GLOBALCONSTANTS DefaultPool_PI_Bargraph (* Bargraph geometry and scale constants (Length, ScalePx, Min, Max, Type) *)
  PACKAGE Uebungen::const::UT::PI;
  VAR_GLOBAL CONSTANT
    Bargraph_PI_I01_ScalePx : REAL := 4.68;
    Bargraph_PI_I01_LengthPx : REAL := 468.0;
    Bargraph_PI_I01_Min : REAL := 0.0;
    Bargraph_PI_I01_Max : REAL := 100.0;
    Bargraph_PI_I01_Type : USINT := 3;
    Bargraph_PI_I02_ScalePx : REAL := 4.68;
    Bargraph_PI_I02_LengthPx : REAL := 468.0;
    Bargraph_PI_I02_Min : REAL := 0.0;
    Bargraph_PI_I02_Max : REAL := 100.0;
    Bargraph_PI_I02_Type : USINT := 3;
    Bargraph_PI_I03_ScalePx : REAL := 4.68;
    Bargraph_PI_I03_LengthPx : REAL := 468.0;
    Bargraph_PI_I03_Min : REAL := 0.0;
    Bargraph_PI_I03_Max : REAL := 100.0;
    Bargraph_PI_I03_Type : USINT := 3;
    Bargraph_PI_I04_ScalePx : REAL := 4.68;
    Bargraph_PI_I04_LengthPx : REAL := 468.0;
    Bargraph_PI_I04_Min : REAL := 0.0;
    Bargraph_PI_I04_Max : REAL := 100.0;
    Bargraph_PI_I04_Type : USINT := 3;
    Bargraph_PI_I05_ScalePx : REAL := 4.68;
    Bargraph_PI_I05_LengthPx : REAL := 468.0;
    Bargraph_PI_I05_Min : REAL := 0.0;
    Bargraph_PI_I05_Max : REAL := 100.0;
    Bargraph_PI_I05_Type : USINT := 3;
    Bargraph_PI_I06_ScalePx : REAL := 4.68;
    Bargraph_PI_I06_LengthPx : REAL := 468.0;
    Bargraph_PI_I06_Min : REAL := 0.0;
    Bargraph_PI_I06_Max : REAL := 100.0;
    Bargraph_PI_I06_Type : USINT := 3;
    Bargraph_PI_I07_ScalePx : REAL := 4.68;
    Bargraph_PI_I07_LengthPx : REAL := 468.0;
    Bargraph_PI_I07_Min : REAL := 0.0;
    Bargraph_PI_I07_Max : REAL := 100.0;
    Bargraph_PI_I07_Type : USINT := 3;
    Bargraph_PI_I08_ScalePx : REAL := 4.68;
    Bargraph_PI_I08_LengthPx : REAL := 468.0;
    Bargraph_PI_I08_Min : REAL := 0.0;
    Bargraph_PI_I08_Max : REAL := 100.0;
    Bargraph_PI_I08_Type : USINT := 3;
  END_VAR
END_GLOBALCONSTANTS
